KUKA KRL program: EHACalib.src, EHACalib.dat

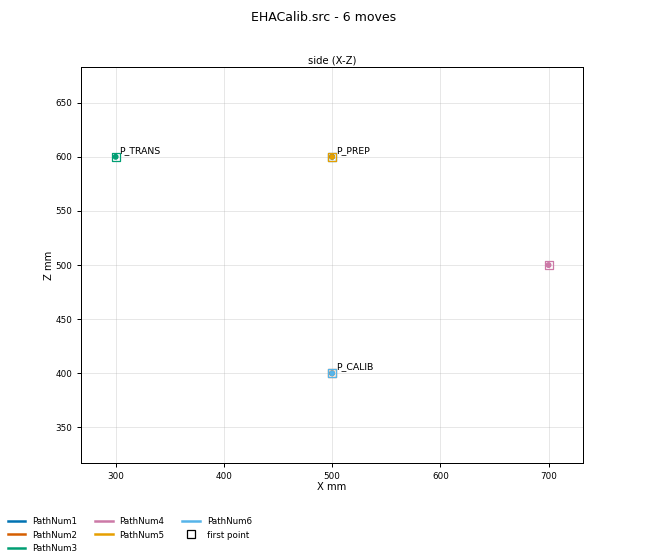
[picture p0: tool path of EHACalib.src, 6 of 12 moves have a stored position in this frame; points joined in program order, loops and branches not executed]
--- EHACalib.src ---
&ACCESS RVP
&REL 1
&PARAM EDITMASK = *
&COMMENT EHA标定系统 - 机器人主程序

; ============================================================================
; 文件说明
;   部署位置 ： KRC:\R1\Program\EHACalib\
;   同目录文件： EHACalib.dat
;   EKI 配置  ： BINKKR.xml（Port 56001，命令接收）
;   Submit   ： BINKKS.sub（Port 56000，状态上报，需配置为 Submit 自启动）
;
; 路径点（在 EHACalib.dat 中修改，示教后替换占位坐标）：
;   PathNum1 → P_PREP  : 预备点（竖直，不接触传感器）
;   PathNum2 → P_CALIB : 标定接触点（EHA 接触力传感器，位移零点）
;   PathNum3 → P_TRANS : 过渡点（安全收回到水平前）
;   PathNum4 → P_LEVEL : 水平姿态（力矩清零位）
;   PathNum5 → P_MASS  : 质量补偿点（竖直，自重调零）
;   PathNum6 → P_TEST  : 检测接触点（输出力检测）
; ============================================================================

DEF EHACalib()

   ;FOLD INI
      ;FOLD BASISTECH INI
         GLOBAL INTERRUPT DECL 3 WHEN $STOPMESS==TRUE DO IR_STOPM()
         INTERRUPT ON 3
         BAS(#INITMOV, 0)
      ;ENDFOLD (BASISTECH INI)
   ;ENDFOLD (INI)

   BAS(#INITMOV, 0)

   ; 初始化 EKI 命令通道并回到当前位置
   BINKKR_INIT()

   CONTINUE
   CYCLE:
   BINKKR_GET()

   IF CONTROL_TYPE_GET == 0 THEN      ; kConfig：触发路径程序 / 外设控制
      PathJob()
      PCJob()
   ELSE
      IF CONTROL_TYPE_GET == 1 THEN   ; kMoving：单点运动
         BINKKRMOVE()
      ENDIF
   ENDIF

   GOTO CYCLE

END

; ── BINKKR_INIT：初始化 EKI 命令通道 ─────────────────────────────────────────
DEF BINKKR_INIT()
   DECL INT I

   POS_TGT_CARTESIUS = $POS_ACT_MES
   POS_CMD_CARTESIUS = POS_TGT_CARTESIUS
   POS_TGT_AXIS = $AXIS_ACT_MEAS
   POS_CMD_AXIS = POS_TGT_AXIS
   CONTINUE
   PTP POS_TGT_AXIS

   FOR I = 1 TO 64
      Bytes[I] = 0
   ENDFOR

   ; 初始化多点路径缓存（与参考工程一致）
   FOR POSNUM = 1 TO 1000 STEP 1
      POINTS[POSNUM] = NULLPOINT
   ENDFOR

   CONNECT:
   EKI_RET = EKI_INIT("BINKKR")
   EKI_RET = EKI_OPEN("BINKKR")
   IF (NOT EKI_RET.CONNECTED) OR ($ERR.NUMBER > 0) THEN
      EKI_RET = EKI_CLOSE("BINKKR")
      EKI_RET = EKI_CLEAR("BINKKR")
      ERR_RAISE($ERR)
      WAIT SEC 2
      GOTO CONNECT
   ENDIF

END

; ── BINKKR_GET：阻塞等待并解析命令包 ─────────────────────────────────────────
DEF BINKKR_GET()
   WAIT SEC 0.0

   WAIT_Flag:
   TimerAction(#TimerStart, 64, -1)
   WAIT FOR ($FLAG[2] OR ($TIMER[64] >= 3000))
   ON_ERROR_PROCEED
   EKI_RET = EKI_GetString("BINKKR", "RcvBuffer", Bytes[])
   TimerAction(#TimerStop, 64, -1)

   IF NOT EKI_RET.Connected THEN
      BINKKR_INIT()
      GOTO WAIT_Flag
   ELSE
      IF NOT $FLAG[2] THEN
         GOTO WAIT_Flag
      ENDIF
   ENDIF
   $FLAG[2] = FALSE

   ; 重置所有解析变量（与参考工程完全一致）
   CONTROL_TYPE_GET    = -1
   MOVING_TYPE_GET     = -1
   COORDINATE_TYPE_GET = -1
   TOOL_NUM            = -1
   Path_NUM            = -1
   READSUCESS          = FALSE
   REVPOSLENGTH        = -1
   RECVDONE            = FALSE
   ControlValve        = -1
   SETSPEED[1]         = -1
   SETSPEED[2]         = -1
   SETSPEED[3]         = -1
   SETSPEED[4]         = -1
   POS_CMD_CARTESIUS.X = -1
   POS_CMD_CARTESIUS.Y = -1
   POS_CMD_CARTESIUS.Z = -1
   POS_CMD_AXIS        = NULLAXIS

   ; 解析命令包
   OFFSET = 0
   CAST_FROM(Bytes[], OFFSET, RCVPOS[], RCVChars[], ReadSPEED, REVPOSLENGTH)
   $VEL.CP             = ReadSPEED
   CONTROL_TYPE_GET    = RCVChars[1]   ; byte[24]
   MOVING_TYPE_GET     = RCVChars[2]   ; byte[25]
   COORDINATE_TYPE_GET = RCVChars[3]   ; byte[26]
   ;$ADVANCE            = RCVChars[4]   ; byte[27]
   $ADVANCE            = 5
   $OV_PRO             = RCVChars[5]   ; byte[28]
   TOOL_NUM            = RCVChars[6]   ; byte[29]
   Path_NUM            = RCVChars[7]   ; byte[30]
   $TOOL               = TOOL_DATA[TOOL_NUM]   ; 直接赋值，上位机保证 TOOL_NUM 有效
   $ACT_TOOL           = TOOL_NUM
   ControlValve        = RCVChars[8]   ; byte[31]

   ; 填充目标坐标（与参考工程 SWITCH/CASE 结构一致）
   SWITCH COORDINATE_TYPE_GET
      CASE 0   ; 笛卡尔坐标
         SWITCH MOVING_TYPE_GET
            CASE 0, 1, 2, 3   ; 单点运动
               POS_CMD_CARTESIUS.X = RCVPOS[1]
               POS_CMD_CARTESIUS.Y = RCVPOS[2]
               POS_CMD_CARTESIUS.Z = RCVPOS[3]
               POS_CMD_CARTESIUS.A = RCVPOS[4]
               POS_CMD_CARTESIUS.B = RCVPOS[5]
               POS_CMD_CARTESIUS.C = RCVPOS[6]
            CASE 4, 5, 6   ; 多点路径（逐包接收，本项目暂不使用）
               POSNUM = 1
               IF REVPOSLENGTH < 1 THEN
                  RECVDONE = FALSE
                  GOTO CLEAR
               ENDIF
               POS_CMD_CARTESIUS.X = RCVPOS[1]
               POS_CMD_CARTESIUS.Y = RCVPOS[2]
               POS_CMD_CARTESIUS.Z = RCVPOS[3]
               POS_CMD_CARTESIUS.A = RCVPOS[4]
               POS_CMD_CARTESIUS.B = RCVPOS[5]
               POS_CMD_CARTESIUS.C = RCVPOS[6]
               POINTS[POSNUM] = POS_CMD_CARTESIUS
               POSNUM = 2
               WHILE POSNUM <= REVPOSLENGTH
                  IF (POSNUM < 5) THEN
                     SETSPEED[POSNUM - 1] = ReadSPEED
                  ENDIF
                  EKI_RET = EKI_Send("BINKKR", Bytes[])
                  WAIT SEC 0.0
                  WAIT FOR $FLAG[2]
                  EKI_RET = EKI_GetString("BINKKR", "RcvBuffer", Bytes[])
                  $FLAG[2] = FALSE
                  OFFSET = 0
                  CAST_FROM(Bytes[], OFFSET, RCVPOS[], RCVChars[], ReadSPEED, REVPOSLENGTH)
                  POS_CMD_CARTESIUS.X = RCVPOS[1]
                  POS_CMD_CARTESIUS.Y = RCVPOS[2]
                  POS_CMD_CARTESIUS.Z = RCVPOS[3]
                  POS_CMD_CARTESIUS.A = RCVPOS[4]
                  POS_CMD_CARTESIUS.B = RCVPOS[5]
                  POS_CMD_CARTESIUS.C = RCVPOS[6]
                  POINTS[POSNUM] = POS_CMD_CARTESIUS
                  POSNUM = POSNUM + 1
               ENDWHILE
         ENDSWITCH

      CASE 1   ; 轴坐标
         POS_CMD_AXIS.A1 = RCVPOS[1]
         POS_CMD_AXIS.A2 = RCVPOS[2]
         POS_CMD_AXIS.A3 = RCVPOS[3]
         POS_CMD_AXIS.A4 = RCVPOS[4]
         POS_CMD_AXIS.A5 = RCVPOS[5]
         POS_CMD_AXIS.A6 = RCVPOS[6]

      DEFAULT
   ENDSWITCH

   RECVDONE = TRUE
   EKI_RET = EKI_Send("BINKKR", Bytes[])   ; 发送 ACK

   CLEAR:
   WAIT SEC 0

END

; ── BINKKRMOVE：执行单点/多点运动 ────────────────────────────────────────────
DEF BINKKRMOVE()
   IF NOT RECVDONE THEN RETURN ENDIF

   POS_CMD_CARTESIUS.S = $POS_ACT_MES.S
   POS_CMD_CARTESIUS.T = $POS_ACT_MES.T

   SWITCH COORDINATE_TYPE_GET
      CASE 0   ; 笛卡尔
         SWITCH MOVING_TYPE_GET
            CASE 0 : LIN POS_CMD_CARTESIUS
            CASE 1 : PTP POS_CMD_CARTESIUS
            CASE 2 : LIN_REL POS_CMD_CARTESIUS #TOOL
            CASE 3 : PTP_REL POS_CMD_CARTESIUS #TOOL
            CASE 4   ; 多点直线路径
               $APO.CDIS = 10
               $VEL.CP = SETSPEED[1]
               LIN POINTS[1] C_DIS C_Dis
               LIN POINTS[2] C_DIS C_Dis
               FOR POSNUM = 3 TO REVPOSLENGTH-1 STEP 1
                  $VEL.CP = SETSPEED[2]
                  LIN POINTS[POSNUM] C_DIS C_Dis
               ENDFOR
               $VEL.CP = SETSPEED[3]
               LIN POINTS[REVPOSLENGTH] C_DIS C_Dis
            DEFAULT
         ENDSWITCH
      CASE 1   ; 轴坐标
         PTP POS_CMD_AXIS C_PTP
      DEFAULT
   ENDSWITCH
END

; ── PathJob：路径程序分发（CASE 0 保留与参考工程一致）────────────────────────
DEF PathJob()
   SWITCH Path_NUM
      CASE 0
         ; 无操作
      CASE 1 : PathNum1()   ; 预备点
      CASE 2 : PathNum2()   ; 标定接触点
      CASE 3 : PathNum3()   ; 过渡点
      CASE 4 : PathNum4()   ; 水平姿态（力矩清零位）
      CASE 5 : PathNum5()   ; 质量补偿点
      CASE 6 : PathNum6()   ; 检测接触点
      DEFAULT
   ENDSWITCH
END

; ── PCJob：外设控制（本项目无外设，ControlValve<0 直接返回）─────────────────
DEF PCJob()
   IF ControlValve < 0 THEN
      RETURN
   ENDIF
   ; 如需扩展 IO 控制，在此添加 SWITCH ControlValve CASE ...
END

; ── EKI_RESET：紧急重置通道（供调试用）──────────────────────────────────────
DEF EKI_RESET()
   EKI_RET = EKI_CLEAR("BINKKR")
   EKI_RET = EKI_INIT("BINKKR")
   EKI_RET = EKI_OPEN("BINKKR")
END

; ============================================================================
; 路径子程序
; ⚠ 以下点位坐标为占位符，必须在示教器示教后修改 EHACalib.dat 中的 P_xxx
; ============================================================================

; PATH1：预备点 ─ 竖直姿态，EHA 不接触力传感器
DEF PathNum1()
   $VEL.CP = 0.1
   PTP P_PREP
END

; PATH2：标定接触点 ─ EHA 接触力传感器，位移零点附近
DEF PathNum2()
   $VEL.CP = 0.05
   LIN P_CALIB
END

; PATH3：过渡点 ─ 从标定点安全收回
DEF PathNum3()
   $VEL.CP = 0.1
   LIN P_TRANS
END

; PATH4：水平姿态 ─ 力矩清零位置
DEF PathNum4()
   $VEL.CP = 0.05
   PTP P_LEVEL
END

; PATH5：质量补偿点 ─ 竖直姿态，自重补偿调零
DEF PathNum5()
   $VEL.CP = 0.1
   PTP P_MASS
END

; PATH6：检测接触点 ─ 输出力检测
DEF PathNum6()
   $VEL.CP = 0.05
   LIN P_TEST
END

--- EHACalib.dat ---
&ACCESS RVP
&REL 1
&PARAM DISKPATH = KRC:\R1\EHACalib
DEFDAT EHACalib PUBLIC

; ── 外部声明（与参考 Main.dat 结构一致）──────────────────────────────────────
EXT BAS (BAS_COMMAND :IN, REAL :IN)
DECL INT SUCCESS

; ── EKI 通讯变量 ──────────────────────────────────────────────────────────────
DECL CHAR       Bytes[64]
DECL INT        OFFSET
DECL EKI_STATUS EKI_RET
DECL REAL       RCVPOS[6]
DECL CHAR       RCVChars[8]
DECL REAL       ReadSPEED

; ── 命令解析结果 ──────────────────────────────────────────────────────────────
DECL INT  CONTROL_TYPE_GET
DECL INT  MOVING_TYPE_GET
DECL INT  COORDINATE_TYPE_GET
DECL INT  TOOL_NUM
DECL INT  Path_NUM
DECL INT  ControlValve
DECL BOOL RECVDONE
DECL BOOL READSUCESS = FALSE

; ── 多点路径变量 ──────────────────────────────────────────────────────────────
DECL INT   POSNUM
DECL INT   REVPOSLENGTH
DECL REAL  SETSPEED[4]
DECL E6POS POINTS[1000]

; ── 运动目标（E6POS / E6AXIS，与参考 Main.dat 类型完全一致）──────────────────
DECL E6POS POS_TGT_CARTESIUS
DECL E6POS POS_CMD_CARTESIUS = {X 0.0, Y 0.0, Z 0.0, A 0.0, B 0.0, C 0.0, S 'B0010', T 'B00101010', E1 0.0, E2 0.0, E3 0.0, E4 0.0, E5 0.0, E6 0.0}
DECL E6AXIS POS_TGT_AXIS
DECL AXIS  POS_CMD_AXIS = {A1 -1.0, A2 -1.0, A3 -1.0, A4 -1.0, A5 -1.0, A6 -1.0}

; ── 空值常量（与参考 Main.dat 完全一致）──────────────────────────────────────
DECL E6POS NULLPOINT = {X -1.0, Y -1.0, Z -1.0, A -1.0, B -1.0, C -1.0, S 'B0010', T 'B0010', E1 0.0, E2 0.0, E3 0.0, E4 0.0, E5 0.0, E6 0.0}
DECL AXIS  NULLAXIS  = {A1 -1.0, A2 -1.0, A3 -1.0, A4 -1.0, A5 -1.0, A6 -1.0}

; ── 标定路径点位 ──────────────────────────────────────────────────────────────
; ⚠ 以下坐标为占位符，必须在示教器上示教真实点位后替换
; PATH1：预备点（竖直姿态，EHA 不接触力传感器）
DECL E6POS P_PREP  = {X 500.0, Y 0.0, Z 600.0, A 0.0, B 0.0, C 0.0, S 2, T 35, E1 0.0, E2 0.0, E3 0.0, E4 0.0, E5 0.0, E6 0.0}

; PATH2：标定接触点（EHA 接触力传感器，位移零点附近）
DECL E6POS P_CALIB = {X 500.0, Y 0.0, Z 400.0, A 0.0, B 0.0, C 0.0, S 2, T 35, E1 0.0, E2 0.0, E3 0.0, E4 0.0, E5 0.0, E6 0.0}

; PATH3：过渡点（从标定点安全收回，向水平姿态过渡）
DECL E6POS P_TRANS = {X 300.0, Y 0.0, Z 600.0, A 0.0, B 0.0, C 0.0, S 2, T 35, E1 0.0, E2 0.0, E3 0.0, E4 0.0, E5 0.0, E6 0.0}

; PATH4：水平姿态点（力矩清零，EHA 轴线水平）
DECL E6POS P_LEVEL = {X 700.0, Y 0.0, Z 500.0, A 0.0, B 90.0, C 0.0, S 2, T 35, E1 0.0, E2 0.0, E3 0.0, E4 0.0, E5 0.0, E6 0.0}

; PATH5：质量补偿点（竖直姿态，自重补偿调零）
DECL E6POS P_MASS  = {X 500.0, Y 0.0, Z 600.0, A 0.0, B 0.0, C 0.0, S 2, T 35, E1 0.0, E2 0.0, E3 0.0, E4 0.0, E5 0.0, E6 0.0}

; PATH6：检测接触点（与力传感器接触，输出力检测）
DECL E6POS P_TEST  = {X 500.0, Y 0.0, Z 400.0, A 0.0, B 0.0, C 0.0, S 2, T 35, E1 0.0, E2 0.0, E3 0.0, E4 0.0, E5 0.0, E6 0.0}

ENDDAT
